// global function to extract e_progress from combined value
FUNCTION f_GetProgress : uint
VAR_INPUT
  state     : UINT;
END_VAR
VAR
  nP        : uint;
END_VAR


nP := state / E_PROGRESS.PROGRESS_INIT;

f_GetProgress := nP * E_PROGRESS.PROGRESS_INIT;

END_FUNCTION

(* stored: Version 1.1.0.1
   POU f_GetProgress: Id {b04d1371-58c5-4697-9b80-ccdeece26464}, SpecialFunc None *)
